// TIA Portal project "AMATROL STATION 1" (V16)

(* hardware
DEVICE "S7300/ET200M station_1"  S7-300 station
   slot 0: "Rail_0"  Rail  6ES7 390-1***0-0AA0
   slot 2: "PLC_1"  CPU 314C-2 DP  6ES7 314-6CH04-0AB0  V3.3
      slot 0: "MPI interface_1"  MPI
      slot 1: "DP interface_1"  DP
      slot 2: "DI 24/DO 16_1"  DI24/DO16
      slot 3: "AI 5/AO 2_1"  AI5/AO2
      slot 4: "Count_1"  Counter
      slot 5: "Positioning_1"  Positioning
*)

// ===== PLC "PLC_1"  CPU 314C-2 DP =====

VAR_GLOBAL   // PLC tag table "INPUTS AND OUTPUTS"
   "S3_Start" AT %I0.0 : Bool;   // Start Button
   "S4_Stop_Button" AT %I0.1 : Bool;   // Stop Button
   "S5_Emergency_Stop" AT %I0.2 : Bool;   // Emergency Stop
   "S2_Output_Power" AT %I0.3 : Bool;   // Output Power
   "IN1_PREV" AT %I0.4 : Bool;
   "IN2_PREV" AT %I0.5 : Bool;
   "IN1_NEXT" AT %I0.6 : Bool;
   "IN2_NEXT" AT %I0.7 : Bool;
   "S6_RESET" AT %I1.0 : Bool;
   "S6_AUTO" AT %I1.1 : Bool;
   "1B1_Feed_Cylinder_Retracted" AT %I1.2 : Bool;   // Feed Cylinder Retracted
   "1B2_Feed_Cylinder_Extended" AT %I1.3 : Bool;   // Feed Cylinder Extended
   "3B1_Pick_Up_Retracted" AT %I1.4 : Bool;   // Pick up retracted
   "3B2_Pick_Up_Extended" AT %I1.5 : Bool;
   "4B1_traverse_retracted" AT %I2.0 : Bool;   // Linear Traverse Cylinder 4A retracted
   "4B2_traverse_extended" AT %I2.1 : Bool;   // Linear Traverse Cylinder 4A extended
   "2P1_Vacuum_ON" AT %I2.6 : Bool;   // Vacuum ON
   "B1_Body Present" AT %I2.7 : Bool;   // Body Present In Feeder Magazine
   "H3_AUTOMATIC_ON_Green" AT %Q4.0 : Bool;
   "OUT1_PREV" AT %Q4.1 : Bool;
   "OUT2_PREV" AT %Q4.2 : Bool;
   "OUT1_NEXT" AT %Q4.3 : Bool;
   "OUT2_NEXT" AT %Q4.4 : Bool;
   "1M1_1A" AT %Q4.5 : Bool;   // Extend Feed Cylinder
   "3M1_3A" AT %Q4.6 : Bool;   // Extend Pick_Up cylinder
   "3M2" AT %Q4.7 : Bool;   // Retract Pick_Up cylinder
   "2M1" AT %Q5.3 : Bool;   // Vacuum Generator ON
   "2M2" AT %Q5.4 : Bool;   // Vacuum Generator OFF
   "4M2" AT %Q5.5 : Bool;   // Retract Linear Traverse Cylinder
   "4M1" AT %Q5.6 : Bool;   // Extend Linear Traverse Cylinder
   "Clock_Memory" AT %M0.1 : Bool;
   "MEM" AT %M0.2 : Bool;
   "AUTO_MODE" AT %Q5.7 : Bool;
   "STOP_MEMORY" AT %M0.3 : Bool;
   "AUTOMODE_MEM" AT %M0.4 : Bool;
END_VAR

DATA_BLOCK "STEPS"   // DB1
{ S7_Optimized_Access := 'FALSE' }
VERSION : 0.1
   VAR
      Current_Step : Int := 0;   // This indicates the step will are currently in
   END_VAR
BEGIN
END_DATA_BLOCK

ORGANIZATION_BLOCK "Main"   // OB1, LAD
TITLE = "Main Program Sweep (Cycle)"
{ S7_Optimized_Access := 'FALSE' }
VERSION : 0.1
   VAR_TEMP
      OB1_EV_CLASS : Byte;   // Bits 0-3 = 1 (Coming event), Bits 4-7 = 1 (Event class 1)
      OB1_SCAN_1 : Byte;   // 1 (Cold restart scan 1 of OB 1), 3 (Scan 2-n of OB 1)
      OB1_PRIORITY : Byte;   // Priority of OB Execution
      OB1_OB_NUMBR : Byte;   // 1 (Organization block 1, OB1)
      OB1_RESERVED_1 : Byte;   // Reserved for system
      OB1_RESERVED_2 : Byte;   // Reserved for system
      OB1_PREV_CYCLE : Int;   // Cycle time of previous OB1 scan (milliseconds)
      OB1_MIN_CYCLE : Int;   // Minimum cycle time of OB1 (milliseconds)
      OB1_MAX_CYCLE : Int;   // Maximum cycle time of OB1 (milliseconds)
      OB1_DATE_TIME : Date_And_Time;   // Date and time OB1 started
   END_VAR
   VAR_TEMP   // added for the SCL form of the ladder/FBD networks
      _w1 : Bool;
   END_VAR
BEGIN

REGION Network 1
   // z
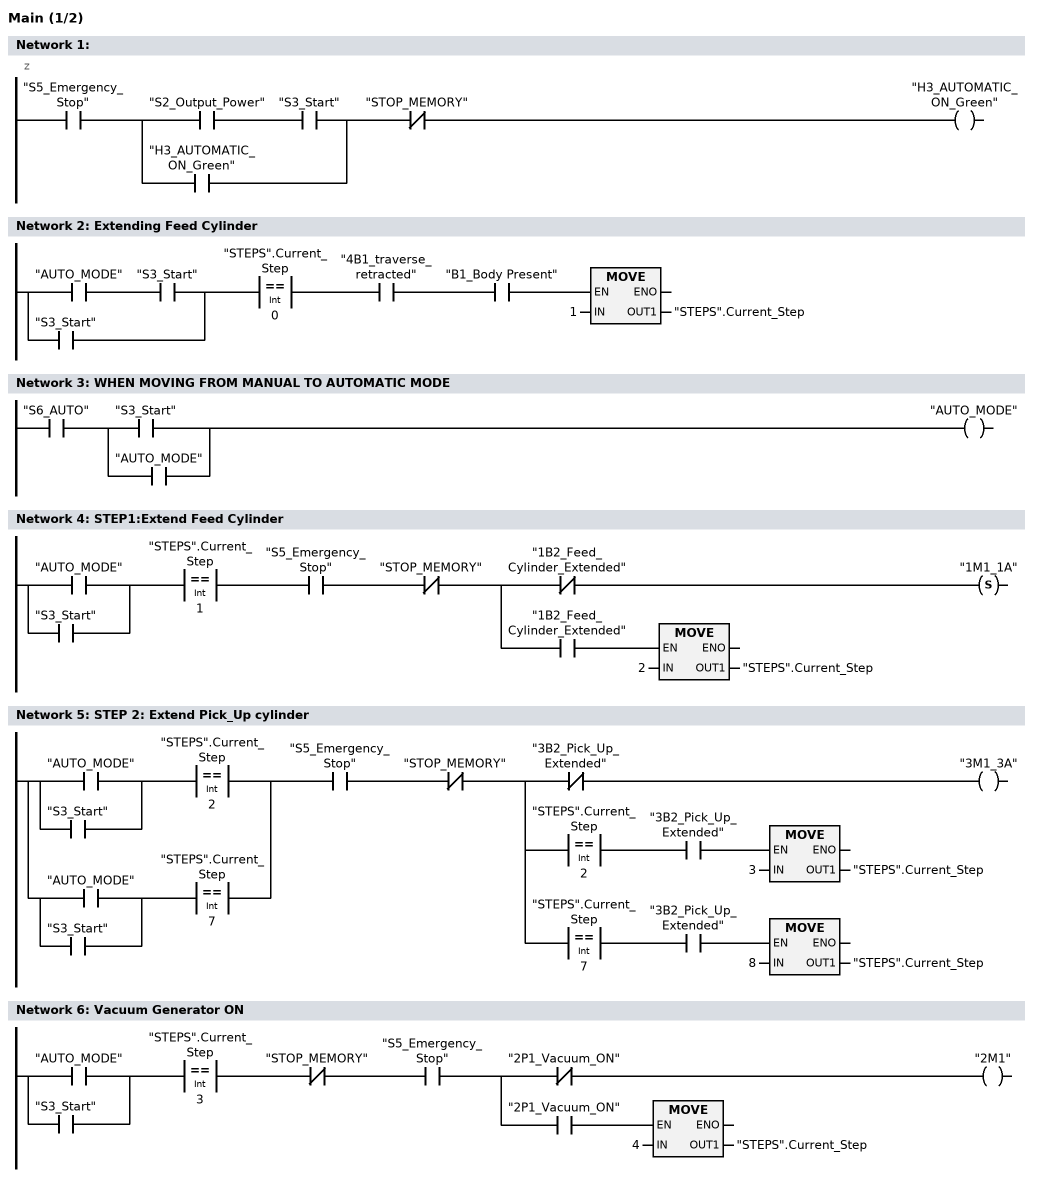
   RUNG wire#powerrail
      Contact( "S5_Emergency_Stop" )
      wire#w1
      Contact( "S2_Output_Power" )
      Contact( "S3_Start" )
      wire#w2
      I_Contact( "STOP_MEMORY" )
      Coil( "H3_AUTOMATIC_ON_Green" )
   END_RUNG
   RUNG wire#w1
      Contact( "H3_AUTOMATIC_ON_Green" )
   END_RUNG wire#w2
   // the same network as SCL:
   "H3_AUTOMATIC_ON_Green" := "S5_Emergency_Stop" AND (("S2_Output_Power" AND "S3_Start") OR "H3_AUTOMATIC_ON_Green") AND NOT "STOP_MEMORY";
END_REGION

REGION Network 2: Extending Feed Cylinder
   RUNG wire#powerrail
      Contact( "AUTO_MODE" )
      Contact( "S3_Start" )
      wire#w1
      { S7_Templates := "SrcType := Int" } EQ_Contact(in1 := "STEPS".Current_Step, in2 := 0)
      Contact( "4B1_traverse_retracted" )
      Contact( "B1_Body Present" )
      { S7_GenerateENO := "TRUE" } Move(in := 1, out1 => "STEPS".Current_Step)
   END_RUNG
   RUNG wire#powerrail
      Contact( "S3_Start" )
   END_RUNG wire#w1
   // the same network as SCL:
   IF (("AUTO_MODE" AND "S3_Start") OR "S3_Start") AND ("STEPS".Current_Step = 0) AND "4B1_traverse_retracted" AND "B1_Body Present" THEN
       "STEPS".Current_Step := 1;
   END_IF;
END_REGION

REGION Network 3: WHEN MOVING FROM MANUAL TO AUTOMATIC MODE
   RUNG wire#powerrail
      Contact( "S6_AUTO" )
      wire#w1
      Contact( "S3_Start" )
      wire#w2
      Coil( "AUTO_MODE" )
   END_RUNG
   RUNG wire#w1
      Contact( "AUTO_MODE" )
   END_RUNG wire#w2
   // the same network as SCL:
   "AUTO_MODE" := "S6_AUTO" AND ("S3_Start" OR "AUTO_MODE");
END_REGION

REGION Network 4: STEP1:Extend Feed Cylinder
   RUNG wire#powerrail
      Contact( "AUTO_MODE" )
      wire#w1
      { S7_Templates := "SrcType := Int" } EQ_Contact(in1 := "STEPS".Current_Step, in2 := 1)
      Contact( "S5_Emergency_Stop" )
      I_Contact( "STOP_MEMORY" )
      wire#w2
      I_Contact( "1B2_Feed_Cylinder_Extended" )
      S_Coil( "1M1_1A" )
   END_RUNG
   RUNG wire#powerrail
      Contact( "S3_Start" )
   END_RUNG wire#w1
   RUNG wire#w2
      Contact( "1B2_Feed_Cylinder_Extended" )
      { S7_GenerateENO := "TRUE" } Move(in := 2, out1 => "STEPS".Current_Step)
   END_RUNG
   // the same network as SCL:
   #_w1 := ("AUTO_MODE" OR "S3_Start") AND ("STEPS".Current_Step = 1) AND "S5_Emergency_Stop" AND NOT "STOP_MEMORY";
   IF #_w1 AND NOT "1B2_Feed_Cylinder_Extended" THEN "1M1_1A" := TRUE; END_IF;
   IF #_w1 AND "1B2_Feed_Cylinder_Extended" THEN "STEPS".Current_Step := 2; END_IF;
END_REGION

REGION Network 5: STEP 2: Extend Pick_Up cylinder
   RUNG wire#powerrail
      Contact( "AUTO_MODE" )
      wire#w1
      { S7_Templates := "SrcType := Int" } EQ_Contact(in1 := "STEPS".Current_Step, in2 := 2)
      wire#w2
      Contact( "S5_Emergency_Stop" )
      I_Contact( "STOP_MEMORY" )
      wire#w4
      I_Contact( "3B2_Pick_Up_Extended" )
      Coil( "3M1_3A" )
   END_RUNG
   RUNG wire#powerrail
      Contact( "S3_Start" )
   END_RUNG wire#w1
   RUNG wire#powerrail
      Contact( "AUTO_MODE" )
      wire#w3
      { S7_Templates := "SrcType := Int" } EQ_Contact(in1 := "STEPS".Current_Step, in2 := 7)
   END_RUNG wire#w2
   RUNG wire#powerrail
      Contact( "S3_Start" )
   END_RUNG wire#w3
   RUNG wire#w4
      { S7_Templates := "SrcType := Int" } EQ_Contact(in1 := "STEPS".Current_Step, in2 := 2)
      Contact( "3B2_Pick_Up_Extended" )
      { S7_GenerateENO := "TRUE" } Move(in := 3, out1 => "STEPS".Current_Step)
   END_RUNG
   RUNG wire#w4
      { S7_Templates := "SrcType := Int" } EQ_Contact(in1 := "STEPS".Current_Step, in2 := 7)
      Contact( "3B2_Pick_Up_Extended" )
      { S7_GenerateENO := "TRUE" } Move(in := 8, out1 => "STEPS".Current_Step)
   END_RUNG
   // the same network as SCL:
   #_w1 := ((("AUTO_MODE" OR "S3_Start") AND ("STEPS".Current_Step = 2)) OR (("AUTO_MODE" OR "S3_Start") AND ("STEPS".Current_Step = 7))) AND "S5_Emergency_Stop" AND NOT "STOP_MEMORY";
   "3M1_3A" := #_w1 AND NOT "3B2_Pick_Up_Extended";
   IF #_w1 AND ("STEPS".Current_Step = 2) AND "3B2_Pick_Up_Extended" THEN "STEPS".Current_Step := 3; END_IF;
   IF #_w1 AND ("STEPS".Current_Step = 7) AND "3B2_Pick_Up_Extended" THEN "STEPS".Current_Step := 8; END_IF;
END_REGION

REGION Network 6: Vacuum Generator ON
   RUNG wire#powerrail
      Contact( "AUTO_MODE" )
      wire#w1
      { S7_Templates := "SrcType := Int" } EQ_Contact(in1 := "STEPS".Current_Step, in2 := 3)
      I_Contact( "STOP_MEMORY" )
      Contact( "S5_Emergency_Stop" )
      wire#w2
      I_Contact( "2P1_Vacuum_ON" )
      Coil( "2M1" )
   END_RUNG
   RUNG wire#powerrail
      Contact( "S3_Start" )
   END_RUNG wire#w1
   RUNG wire#w2
      Contact( "2P1_Vacuum_ON" )
      { S7_GenerateENO := "TRUE" } Move(in := 4, out1 => "STEPS".Current_Step)
   END_RUNG
   // the same network as SCL:
   #_w1 := ("AUTO_MODE" OR "S3_Start") AND ("STEPS".Current_Step = 3) AND NOT "STOP_MEMORY" AND "S5_Emergency_Stop";
   "2M1" := #_w1 AND NOT "2P1_Vacuum_ON";
   IF #_w1 AND "2P1_Vacuum_ON" THEN "STEPS".Current_Step := 4; END_IF;
END_REGION

REGION Network 7: Retract Feed Cylinder
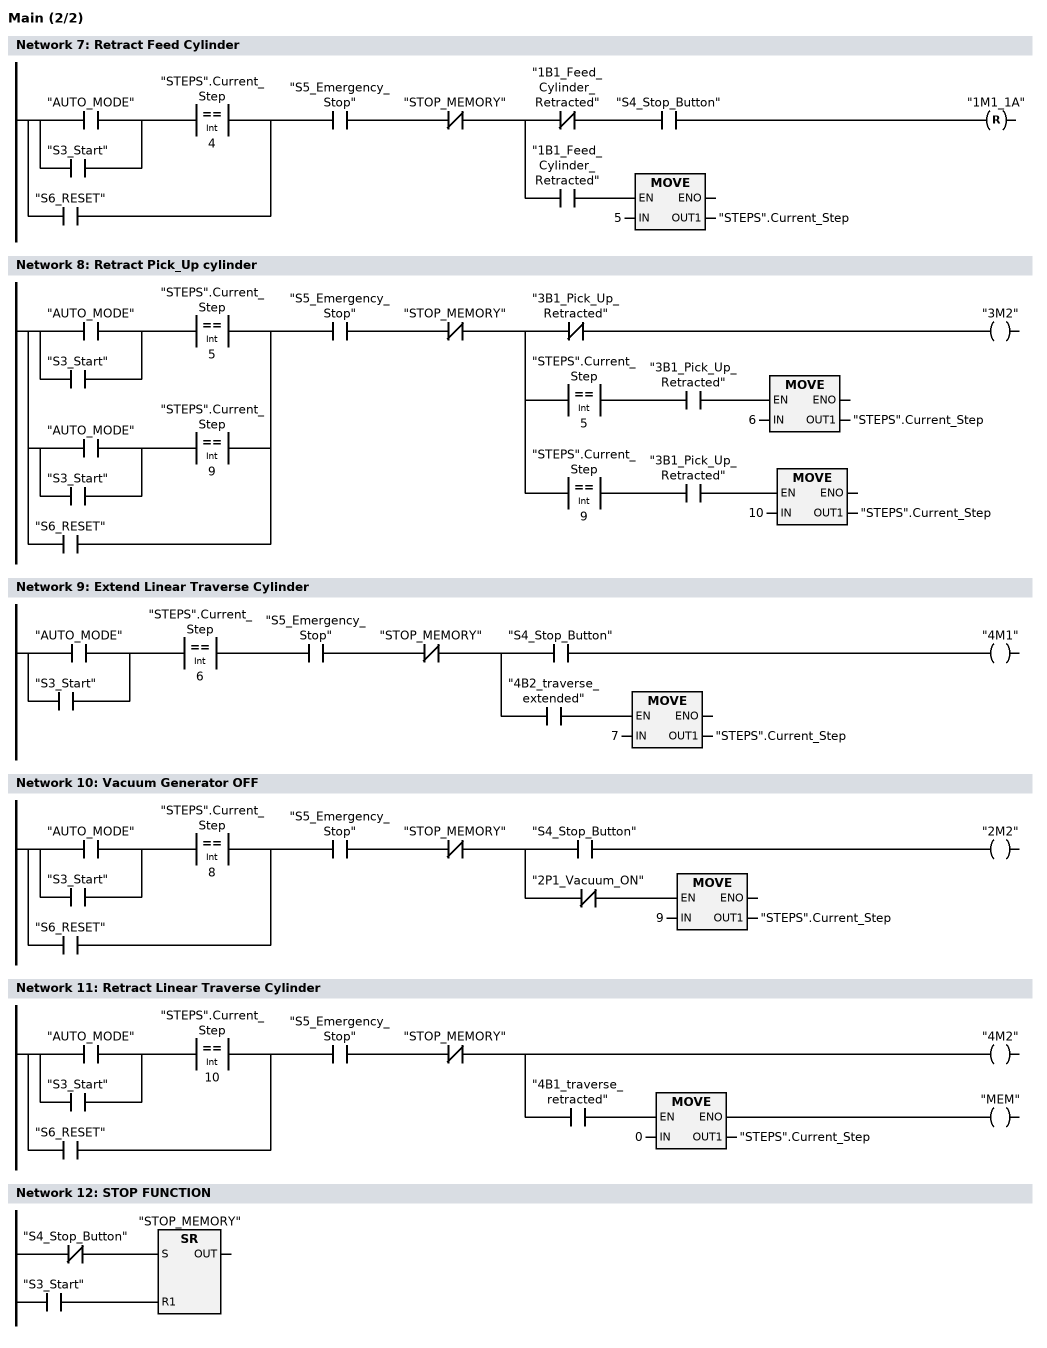
   RUNG wire#powerrail
      Contact( "AUTO_MODE" )
      wire#w1
      { S7_Templates := "SrcType := Int" } EQ_Contact(in1 := "STEPS".Current_Step, in2 := 4)
      wire#w2
      Contact( "S5_Emergency_Stop" )
      I_Contact( "STOP_MEMORY" )
      wire#w3
      I_Contact( "1B1_Feed_Cylinder_Retracted" )
      Contact( "S4_Stop_Button" )
      R_Coil( "1M1_1A" )
   END_RUNG
   RUNG wire#powerrail
      Contact( "S3_Start" )
   END_RUNG wire#w1
   RUNG wire#powerrail
      Contact( "S6_RESET" )
   END_RUNG wire#w2
   RUNG wire#w3
      Contact( "1B1_Feed_Cylinder_Retracted" )
      { S7_GenerateENO := "TRUE" } Move(in := 5, out1 => "STEPS".Current_Step)
   END_RUNG
   // the same network as SCL:
   #_w1 := ((("AUTO_MODE" OR "S3_Start") AND ("STEPS".Current_Step = 4)) OR "S6_RESET") AND "S5_Emergency_Stop" AND NOT "STOP_MEMORY";
   IF #_w1 AND NOT "1B1_Feed_Cylinder_Retracted" AND "S4_Stop_Button" THEN "1M1_1A" := FALSE; END_IF;
   IF #_w1 AND "1B1_Feed_Cylinder_Retracted" THEN "STEPS".Current_Step := 5; END_IF;
END_REGION

REGION Network 8: Retract Pick_Up cylinder
   RUNG wire#powerrail
      Contact( "AUTO_MODE" )
      wire#w1
      { S7_Templates := "SrcType := Int" } EQ_Contact(in1 := "STEPS".Current_Step, in2 := 5)
      wire#w2
      Contact( "S5_Emergency_Stop" )
      I_Contact( "STOP_MEMORY" )
      wire#w4
      I_Contact( "3B1_Pick_Up_Retracted" )
      Coil( "3M2" )
   END_RUNG
   RUNG wire#powerrail
      Contact( "S3_Start" )
   END_RUNG wire#w1
   RUNG wire#powerrail
      Contact( "AUTO_MODE" )
      wire#w3
      { S7_Templates := "SrcType := Int" } EQ_Contact(in1 := "STEPS".Current_Step, in2 := 9)
   END_RUNG wire#w2
   RUNG wire#powerrail
      Contact( "S3_Start" )
   END_RUNG wire#w3
   RUNG wire#powerrail
      Contact( "S6_RESET" )
   END_RUNG wire#w2
   RUNG wire#w4
      { S7_Templates := "SrcType := Int" } EQ_Contact(in1 := "STEPS".Current_Step, in2 := 5)
      Contact( "3B1_Pick_Up_Retracted" )
      { S7_GenerateENO := "TRUE" } Move(in := 6, out1 => "STEPS".Current_Step)
   END_RUNG
   RUNG wire#w4
      { S7_Templates := "SrcType := Int" } EQ_Contact(in1 := "STEPS".Current_Step, in2 := 9)
      Contact( "3B1_Pick_Up_Retracted" )
      { S7_GenerateENO := "TRUE" } Move(in := 10, out1 => "STEPS".Current_Step)
   END_RUNG
   // the same network as SCL:
   #_w1 := ((("AUTO_MODE" OR "S3_Start") AND ("STEPS".Current_Step = 5)) OR (("AUTO_MODE" OR "S3_Start") AND ("STEPS".Current_Step = 9)) OR "S6_RESET") AND "S5_Emergency_Stop" AND NOT "STOP_MEMORY";
   "3M2" := #_w1 AND NOT "3B1_Pick_Up_Retracted";
   IF #_w1 AND ("STEPS".Current_Step = 5) AND "3B1_Pick_Up_Retracted" THEN "STEPS".Current_Step := 6; END_IF;
   IF #_w1 AND ("STEPS".Current_Step = 9) AND "3B1_Pick_Up_Retracted" THEN
       "STEPS".Current_Step := 10;
   END_IF;
END_REGION

REGION Network 9: Extend Linear Traverse Cylinder
   RUNG wire#powerrail
      Contact( "AUTO_MODE" )
      wire#w1
      { S7_Templates := "SrcType := Int" } EQ_Contact(in1 := "STEPS".Current_Step, in2 := 6)
      Contact( "S5_Emergency_Stop" )
      I_Contact( "STOP_MEMORY" )
      wire#w2
      Contact( "S4_Stop_Button" )
      Coil( "4M1" )
   END_RUNG
   RUNG wire#powerrail
      Contact( "S3_Start" )
   END_RUNG wire#w1
   RUNG wire#w2
      Contact( "4B2_traverse_extended" )
      { S7_GenerateENO := "TRUE" } Move(in := 7, out1 => "STEPS".Current_Step)
   END_RUNG
   // the same network as SCL:
   #_w1 := ("AUTO_MODE" OR "S3_Start") AND ("STEPS".Current_Step = 6) AND "S5_Emergency_Stop" AND NOT "STOP_MEMORY";
   "4M1" := #_w1 AND "S4_Stop_Button";
   IF #_w1 AND "4B2_traverse_extended" THEN "STEPS".Current_Step := 7; END_IF;
END_REGION

REGION Network 10: Vacuum Generator OFF
   RUNG wire#powerrail
      Contact( "AUTO_MODE" )
      wire#w1
      { S7_Templates := "SrcType := Int" } EQ_Contact(in1 := "STEPS".Current_Step, in2 := 8)
      wire#w2
      Contact( "S5_Emergency_Stop" )
      I_Contact( "STOP_MEMORY" )
      wire#w3
      Contact( "S4_Stop_Button" )
      Coil( "2M2" )
   END_RUNG
   RUNG wire#powerrail
      Contact( "S3_Start" )
   END_RUNG wire#w1
   RUNG wire#powerrail
      Contact( "S6_RESET" )
   END_RUNG wire#w2
   RUNG wire#w3
      I_Contact( "2P1_Vacuum_ON" )
      { S7_GenerateENO := "TRUE" } Move(in := 9, out1 => "STEPS".Current_Step)
   END_RUNG
   // the same network as SCL:
   #_w1 := ((("AUTO_MODE" OR "S3_Start") AND ("STEPS".Current_Step = 8)) OR "S6_RESET") AND "S5_Emergency_Stop" AND NOT "STOP_MEMORY";
   "2M2" := #_w1 AND "S4_Stop_Button";
   IF #_w1 AND NOT "2P1_Vacuum_ON" THEN "STEPS".Current_Step := 9; END_IF;
END_REGION

REGION Network 11: Retract Linear Traverse Cylinder
   RUNG wire#powerrail
      Contact( "AUTO_MODE" )
      wire#w1
      { S7_Templates := "SrcType := Int" } EQ_Contact(in1 := "STEPS".Current_Step, in2 := 10)
      wire#w2
      Contact( "S5_Emergency_Stop" )
      I_Contact( "STOP_MEMORY" )
      wire#w3
      Coil( "4M2" )
   END_RUNG
   RUNG wire#powerrail
      Contact( "S3_Start" )
   END_RUNG wire#w1
   RUNG wire#powerrail
      Contact( "S6_RESET" )
   END_RUNG wire#w2
   RUNG wire#w3
      Contact( "4B1_traverse_retracted" )
      { S7_GenerateENO := "TRUE" } Move(in := 0, out1 => "STEPS".Current_Step)
      Coil( "MEM" )
   END_RUNG
   // the same network as SCL:
   // ENO of a box is taken as its EN; it also drops when the box reports an error
   "4M2" := ((("AUTO_MODE" OR "S3_Start") AND ("STEPS".Current_Step = 10)) OR "S6_RESET") AND "S5_Emergency_Stop" AND NOT "STOP_MEMORY";
   #_w1 := "4M2" AND "4B1_traverse_retracted";
   IF #_w1 THEN "STEPS".Current_Step := 0; END_IF;
   "MEM" := #_w1;
END_REGION

REGION Network 12: STOP FUNCTION
   RUNG wire#powerrail
      I_Contact( "S4_Stop_Button" )
      S_SR(operand := "STOP_MEMORY", r1 := wire#w1)
   END_RUNG
   RUNG wire#powerrail
      Contact( "S3_Start" )
   END_RUNG wire#w1
   // the same network as SCL:
   IF NOT "S4_Stop_Button" THEN
       "STOP_MEMORY" := TRUE;   // SR flip-flop
   END_IF;
   IF "S3_Start" THEN "STOP_MEMORY" := FALSE; END_IF;
END_REGION
END_ORGANIZATION_BLOCK